PROGRAM p_Regulators
VAR

fbRegProp1	:	FB_ProportionairRegulator;
fbRegProp2	:	FB_ProportionairRegulator;
fbRegProp3	:	FB_ProportionairRegulator;
fbRegProp4	:	FB_ProportionairRegulator;

END_VAR

(* Proportionair regulators *)
fbRegProp1(iq_stRegProp:=stRegProp1);
fbRegProp2(iq_stRegProp:=stRegProp2);
fbRegProp3(iq_stRegProp:=stRegProp3);
fbRegProp4(iq_stRegProp:=stRegProp4);

END_PROGRAM

(* stored: Version 1.1.0.1, ProductVersion 3.1.4020.12
   POU p_Regulators: Id {7fa22113-75a7-40de-8aa7-6bf32b41ae72}, SpecialFunc None *)
